ABB RobotStudio station: Lab1Station.rsstn

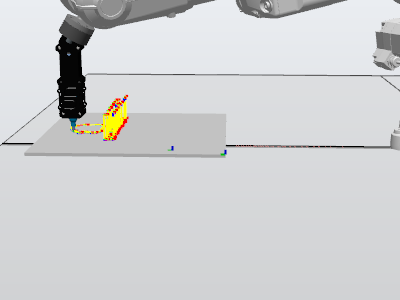
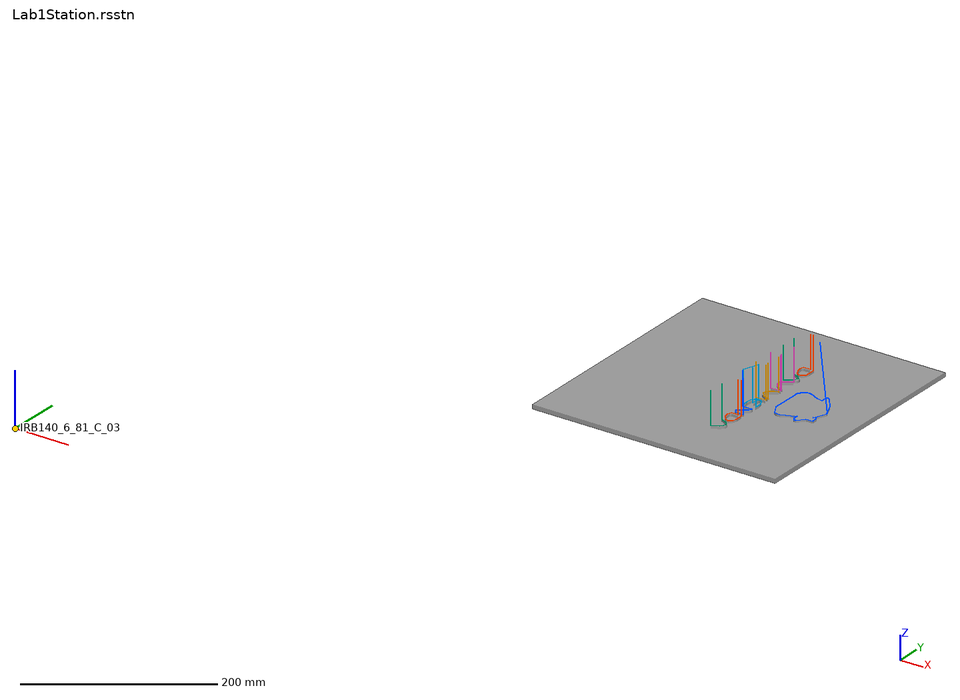
[picture v1: parts stored in the station drawn from their meshes, with robot base, taught points and paths (robot models come from the ABB library and are not in the file)]
Station Lab1Station (saved by RobotStudio 22.3.10190.2)
Controller Controller3
  mechanical unit ROB_1: IRB140_6_81_C_03, 6 joints, base frame (0, 0, 0) mm
Layout (positions relative to the parent item):
  - IRB140_6_81_C_03 [mechanism, from Robots\IRB140_6_81_C_G_03.rslib] at (0, 0, 0) mm; joint values [0.4312, 1.4172, -1.227, -0.2668, 0.9151, 0.5443] (rad or m)
  - HerrMarcador [part, from MyTools\HerrMarcadorInclinado.rslib] at (758.29, 333.88, 278.98) mm, rotated rx -180 ry 30 rz -180 deg
  - Davivienda [part] at (520, 470, 100) mm, rotated rx 0 ry 0 rz -90 deg, size 300 x 300 x 8 mm
Attachment: HerrMarcador is attached to IRB140_6_81_C_03 / Link6
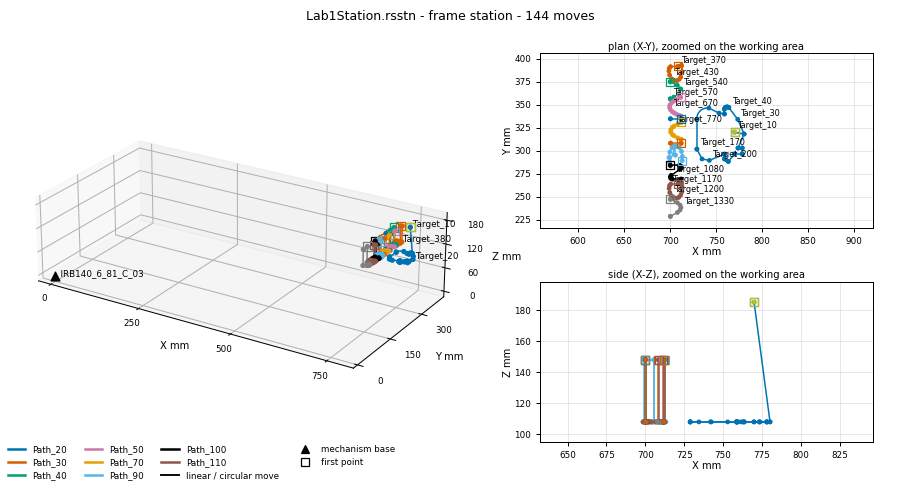
[picture p0: tool path of Lab1Station.rsstn in frame station, 144 of 146 moves have a stored position in this frame; points joined in program order, loops and branches not executed]
Targets, tools, work objects and paths stored in the station, written as RAPID:
! task T_ROB1
MODULE user
  TASK PERS tooldata Marcador_Data:=[TRUE,[[72.5,0,155.57],[0.965925826,-0.000008429,0.258819045,0.000002259]],[0.002,[19.889,-0.005,58.089],[1,0,0,0],0,0,0]];
ENDMODULE

! task T_ROB1
MODULE CalibData
  TASK PERS wobjdata Tablero:=[FALSE,TRUE,"",[[600,450,105],[0.707106781,0,0,-0.707106781]],[[-20,-80,0],[1,0,0,0]]];
ENDMODULE

! task T_ROB1
MODULE Module1
  CONST robtarget Target_10:=[[150,250,80],[0,-0.707106781,0.707106781,0],[0,-1,0,0],[9E+09,9E+09,9E+09,9E+09,9E+09,9E+09]];
  CONST robtarget Target_20:=[[152.02476718,260.252415756,3],[0,-0.707106781,0.707106781,0],[0,-1,1,0],[9E+09,9E+09,9E+09,9E+09,9E+09,9E+09]];
  CONST robtarget Target_30:=[[136.118401169,253.292570976,3],[0,-0.707106781,0.707106781,0],[0,0,0,0],[9E+09,9E+09,9E+09,9E+09,9E+09,9E+09]];
  CONST robtarget Target_40:=[[123.269606583,243.615464733,3],[0,-0.707106781,0.707106781,0],[0,-1,0,0],[9E+09,9E+09,9E+09,9E+09,9E+09,9E+09]];
  CONST robtarget Target_50:=[[123.269606583,243.615464733,3],[0,-0.707106781,0.707106781,0],[0,0,0,0],[9E+09,9E+09,9E+09,9E+09,9E+09,9E+09]];
  CONST robtarget Target_60:=[[122.281773997,241.718097026,3],[0,-0.707106781,0.707106781,0],[0,-1,0,0],[9E+09,9E+09,9E+09,9E+09,9E+09,9E+09]];
  CONST robtarget Target_70:=[[122.995762655,239.701655203,3],[0,-0.707106781,0.707106781,0],[0,0,0,0],[9E+09,9E+09,9E+09,9E+09,9E+09,9E+09]];
  CONST robtarget Target_80:=[[124.957451694,238.84866426,3],[0,-0.707106781,0.707106781,0],[0,0,0,0],[9E+09,9E+09,9E+09,9E+09,9E+09,9E+09]];
  CONST robtarget Target_90:=[[124.957451694,238.84866426,3],[0,-0.707106781,0.707106781,0],[0,0,0,0],[9E+09,9E+09,9E+09,9E+09,9E+09,9E+09]];
  CONST robtarget Target_100:=[[130.248275394,238.84866426,3],[0,-0.707106781,0.707106781,0],[0,0,0,0],[9E+09,9E+09,9E+09,9E+09,9E+09,9E+09]];
  CONST robtarget Target_110:=[[130.248275394,238.84866426,3],[0,-0.707106781,0.707106781,0],[0,0,0,0],[9E+09,9E+09,9E+09,9E+09,9E+09,9E+09]];
  CONST robtarget Target_120:=[[129.335918588,232.983108033,3],[0,-0.707106781,0.707106781,0],[0,0,0,0],[9E+09,9E+09,9E+09,9E+09,9E+09,9E+09]];
  CONST robtarget Target_130:=[[123.812362313,221.9363364,3],[0,-0.707106781,0.707106781,0],[0,0,0,0],[9E+09,9E+09,9E+09,9E+09,9E+09,9E+09]];
  CONST robtarget Target_140:=[[125.443880841,214.375036174,3],[0,-0.707106781,0.707106781,0],[0,0,0,0],[9E+09,9E+09,9E+09,9E+09,9E+09,9E+09]];
  CONST robtarget Target_150:=[[135.991781584,208.907395353,3],[0,-0.707106781,0.707106781,0],[0,0,0,0],[9E+09,9E+09,9E+09,9E+09,9E+09,9E+09]];
  CONST robtarget Target_160:=[[135.991781584,208.907395353,3],[0,-0.707106781,0.707106781,0],[0,0,0,0],[9E+09,9E+09,9E+09,9E+09,9E+09,9E+09]];
  CONST robtarget Target_170:=[[168.476558528,208.907395353,3],[0,-0.707106781,0.707106781,0],[0,0,0,0],[9E+09,9E+09,9E+09,9E+09,9E+09,9E+09]];
  CONST robtarget Target_180:=[[168.476558528,208.907395353,3],[0,-0.707106781,0.707106781,0],[0,0,0,0],[9E+09,9E+09,9E+09,9E+09,9E+09,9E+09]];
  CONST robtarget Target_190:=[[179.114572542,214.493962129,3],[0,-0.707106781,0.707106781,0],[0,0,0,0],[9E+09,9E+09,9E+09,9E+09,9E+09,9E+09]];
  CONST robtarget Target_200:=[[180.686258584,222.455286023,3],[0,-0.707106781,0.707106781,0],[0,0,0,0],[9E+09,9E+09,9E+09,9E+09,9E+09,9E+09]];
  CONST robtarget Target_210:=[[173.93550103,238.84866426,3],[0,-0.707106781,0.707106781,0],[0,0,0,0],[9E+09,9E+09,9E+09,9E+09,9E+09,9E+09]];
  CONST robtarget Target_220:=[[173.93550103,238.84866426,3],[0,-0.707106781,0.707106781,0],[0,0,0,0],[9E+09,9E+09,9E+09,9E+09,9E+09,9E+09]];
  CONST robtarget Target_230:=[[179.092082666,238.84866426,3],[0,-0.707106781,0.707106781,0],[0,0,0,0],[9E+09,9E+09,9E+09,9E+09,9E+09,9E+09]];
  CONST robtarget Target_240:=[[179.092082666,238.84866426,3],[0,-0.707106781,0.707106781,0],[0,0,0,0],[9E+09,9E+09,9E+09,9E+09,9E+09,9E+09]];
  CONST robtarget Target_250:=[[181.598076735,240.213820445,3],[0,-0.707106781,0.707106781,0],[0,0,0,0],[9E+09,9E+09,9E+09,9E+09,9E+09,9E+09]];
  CONST robtarget Target_260:=[[181.810114173,243.059641558,3],[0,-0.707106781,0.707106781,0],[0,0,0,0],[9E+09,9E+09,9E+09,9E+09,9E+09,9E+09]];
  CONST robtarget Target_270:=[[181.810114173,243.059641558,3],[0,-0.707106781,0.707106781,0],[0,0,0,0],[9E+09,9E+09,9E+09,9E+09,9E+09,9E+09]];
  CONST robtarget Target_280:=[[173.790831816,249.924383369,3],[0,-0.707106781,0.707106781,0],[0,0,0,0],[9E+09,9E+09,9E+09,9E+09,9E+09,9E+09]];
  CONST robtarget Target_290:=[[173.790831816,249.924383369,3],[0,-0.707106781,0.707106781,0],[0,0,0,0],[9E+09,9E+09,9E+09,9E+09,9E+09,9E+09]];
  CONST robtarget Target_300:=[[173.790831816,258.182639544,3],[0,-0.707106781,0.707106781,0],[0,0,0,0],[9E+09,9E+09,9E+09,9E+09,9E+09,9E+09]];
  CONST robtarget Target_310:=[[173.790831816,258.182639544,3],[0,-0.707106781,0.707106781,0],[0,0,0,0],[9E+09,9E+09,9E+09,9E+09,9E+09,9E+09]];
  CONST robtarget Target_320:=[[167.241395906,258.182639544,3],[0,-0.707106781,0.707106781,0],[0,0,0,0],[9E+09,9E+09,9E+09,9E+09,9E+09,9E+09]];
  CONST robtarget Target_330:=[[167.241395906,258.182639544,3],[0,-0.707106781,0.707106781,0],[0,0,0,0],[9E+09,9E+09,9E+09,9E+09,9E+09,9E+09]];
  CONST robtarget Target_340:=[[167.241395906,253.645994177,3],[0,-0.707106781,0.707106781,0],[0,0,0,0],[9E+09,9E+09,9E+09,9E+09,9E+09,9E+09]];
  CONST robtarget Target_350:=[[167.241395906,253.645994177,3],[0,-0.707106781,0.707106781,0],[0,0,0,0],[9E+09,9E+09,9E+09,9E+09,9E+09,9E+09]];
  CONST robtarget Target_360:=[[152.02476718,260.252415756,3],[0,-0.707106781,0.707106781,0],[0,0,0,0],[9E+09,9E+09,9E+09,9E+09,9E+09,9E+09]];
  CONST robtarget Target_370:=[[78.556394934,188.285452755,43],[0,-0.707106781,0.707106781,0],[0,0,0,0],[9E+09,9E+09,9E+09,9E+09,9E+09,9E+09]];
  CONST robtarget Target_380:=[[78.556394934,188.285452755,3],[0,-0.707106781,0.707106781,0],[0,0,0,0],[9E+09,9E+09,9E+09,9E+09,9E+09,9E+09]];
  CONST robtarget Target_390:=[[78.777217091,180.337746759,3],[0,-0.707106781,0.707106781,0],[0,0,0,0],[9E+09,9E+09,9E+09,9E+09,9E+09,9E+09]];
  CONST robtarget Target_400:=[[80.371798013,178.989551395,3],[0,-0.707106781,0.707106781,0],[0,0,0,0],[9E+09,9E+09,9E+09,9E+09,9E+09,9E+09]];
  CONST robtarget Target_410:=[[83.506257563,178.489977672,3],[0,-0.707106781,0.707106781,0],[0,0,0,0],[9E+09,9E+09,9E+09,9E+09,9E+09,9E+09]];
  CONST robtarget Target_420:=[[87.997557508,179.252868031,3],[0,-0.707106781,0.707106781,0],[0,0,0,0],[9E+09,9E+09,9E+09,9E+09,9E+09,9E+09]];
  CONST robtarget Target_430:=[[92.028971208,181.53752069,3],[0,-0.707106781,0.707106781,0],[0,0,0,0],[9E+09,9E+09,9E+09,9E+09,9E+09,9E+09]];
  CONST robtarget Target_440:=[[93.868246154,184.336737299,3],[0,-0.707106781,0.707106781,0],[0,0,0,0],[9E+09,9E+09,9E+09,9E+09,9E+09,9E+09]];
  CONST robtarget Target_450:=[[94.007732668,187.144143926,3],[0,-0.707106781,0.707106781,0],[0,0,0,0],[9E+09,9E+09,9E+09,9E+09,9E+09,9E+09]];
  CONST robtarget Target_460:=[[92.604060403,189.719708823,3],[0,-0.707106781,0.707106781,0],[0,0,0,0],[9E+09,9E+09,9E+09,9E+09,9E+09,9E+09]];
  CONST robtarget Target_470:=[[90.06132568,191.417144488,3],[0,-0.707106781,0.707106781,0],[0,0,0,0],[9E+09,9E+09,9E+09,9E+09,9E+09,9E+09]];
  CONST robtarget Target_480:=[[85.079316563,192.471582305,3],[0,-0.707106781,0.707106781,0],[0,0,0,0],[9E+09,9E+09,9E+09,9E+09,9E+09,9E+09]];
  CONST robtarget Target_490:=[[77.598246493,192.118931644,3],[0,-0.707106781,0.707106781,0],[0,0,0,0],[9E+09,9E+09,9E+09,9E+09,9E+09,9E+09]];
  CONST robtarget Target_500:=[[77.598246493,192.118931644,43],[0,-0.707106781,0.707106781,0],[0,0,0,0],[9E+09,9E+09,9E+09,9E+09,9E+09,9E+09]];
  CONST robtarget Target_510:=[[95.28667285,179.972658622,43],[0,-0.707106781,0.707106781,0],[0,0,0,0],[9E+09,9E+09,9E+09,9E+09,9E+09,9E+09]];
  CONST robtarget Target_520:=[[95.28667285,179.972658622,3],[0,-0.707106781,0.707106781,0],[0,0,0,0],[9E+09,9E+09,9E+09,9E+09,9E+09,9E+09]];
  CONST robtarget Target_530:=[[99.054803913,187.648232468,3],[0,-0.707106781,0.707106781,0],[0,0,0,0],[9E+09,9E+09,9E+09,9E+09,9E+09,9E+09]];
  CONST robtarget Target_540:=[[102.919910411,191.254451105,3],[0,-0.707106781,0.707106781,0],[0,0,0,0],[9E+09,9E+09,9E+09,9E+09,9E+09,9E+09]];
  CONST robtarget Target_550:=[[108.350570105,189.25957291,3],[0,-0.707106781,0.707106781,0],[0,0,0,0],[9E+09,9E+09,9E+09,9E+09,9E+09,9E+09]];
  CONST robtarget Target_560:=[[111.949527633,183.734460812,3],[0,-0.707106781,0.707106781,0],[0,0,0,0],[9E+09,9E+09,9E+09,9E+09,9E+09,9E+09]];
  CONST robtarget Target_570:=[[113.857897554,179.972658622,3],[0,-0.707106781,0.707106781,0],[0,0,0,0],[9E+09,9E+09,9E+09,9E+09,9E+09,9E+09]];
  CONST robtarget Target_580:=[[113.857897554,179.972658622,43],[0,-0.707106781,0.707106781,0],[0,0,0,0],[9E+09,9E+09,9E+09,9E+09,9E+09,9E+09]];
  CONST robtarget Target_590:=[[112.126063194,191.2423046,43],[0,-0.707106781,0.707106781,0],[0,0,0,0],[9E+09,9E+09,9E+09,9E+09,9E+09,9E+09]];
  CONST robtarget Target_600:=[[112.126063194,191.2423046,3],[0,-0.707106781,0.707106781,0],[0,0,0,0],[9E+09,9E+09,9E+09,9E+09,9E+09,9E+09]];
  CONST robtarget Target_610:=[[114.401889485,186.789312293,3],[0,-0.707106781,0.707106781,0],[0,0,0,0],[9E+09,9E+09,9E+09,9E+09,9E+09,9E+09]];
  CONST robtarget Target_620:=[[115.58057196,184.74123642,3],[0,-0.707106781,0.707106781,0],[0,0,0,0],[9E+09,9E+09,9E+09,9E+09,9E+09,9E+09]];
  CONST robtarget Target_630:=[[116.864504777,182.854229079,3],[0,-0.707106781,0.707106781,0],[0,0,0,0],[9E+09,9E+09,9E+09,9E+09,9E+09,9E+09]];
  CONST robtarget Target_640:=[[118.25426578,181.252000645,3],[0,-0.707106781,0.707106781,0],[0,0,0,0],[9E+09,9E+09,9E+09,9E+09,9E+09,9E+09]];
  CONST robtarget Target_650:=[[120.57420176,179.604352291,3],[0,-0.707106781,0.707106781,0],[0,0,0,0],[9E+09,9E+09,9E+09,9E+09,9E+09,9E+09]];
  CONST robtarget Target_660:=[[123.164632355,179.201937245,3],[0,-0.707106781,0.707106781,0],[0,0,0,0],[9E+09,9E+09,9E+09,9E+09,9E+09,9E+09]];
  CONST robtarget Target_670:=[[125.643689482,180.211828512,3],[0,-0.707106781,0.707106781,0],[0,0,0,0],[9E+09,9E+09,9E+09,9E+09,9E+09,9E+09]];
  CONST robtarget Target_680:=[[127.787428256,182.296804988,3],[0,-0.707106781,0.707106781,0],[0,0,0,0],[9E+09,9E+09,9E+09,9E+09,9E+09,9E+09]];
  CONST robtarget Target_690:=[[129.053529141,184.108665847,3],[0,-0.707106781,0.707106781,0],[0,0,0,0],[9E+09,9E+09,9E+09,9E+09,9E+09,9E+09]];
  CONST robtarget Target_700:=[[130.193418821,186.12829205,3],[0,-0.707106781,0.707106781,0],[0,0,0,0],[9E+09,9E+09,9E+09,9E+09,9E+09,9E+09]];
  CONST robtarget Target_710:=[[131.496798753,188.892443357,3],[0,-0.707106781,0.707106781,0],[0,0,0,0],[9E+09,9E+09,9E+09,9E+09,9E+09,9E+09]];
  CONST robtarget Target_720:=[[132.509994829,191.333655407,3],[0,-0.707106781,0.707106781,0],[0,0,0,0],[9E+09,9E+09,9E+09,9E+09,9E+09,9E+09]];
  CONST robtarget Target_730:=[[132.509994829,191.333655407,43],[0,-0.707106781,0.707106781,0],[0,0,0,0],[9E+09,9E+09,9E+09,9E+09,9E+09,9E+09]];
  CONST robtarget Target_850:=[[157.76203271,191.808660142,43],[0,-0.707106781,0.707106781,0],[0,0,0,0],[9E+09,9E+09,9E+09,9E+09,9E+09,9E+09]];
  CONST robtarget Target_840:=[[157.76203271,191.808660142,3],[0,-0.707106781,0.707106781,0],[0,0,0,0],[9E+09,9E+09,9E+09,9E+09,9E+09,9E+09]];
  CONST robtarget Target_830:=[[156.15234039,188.046857953,3],[0,-0.707106781,0.707106781,0],[0,0,0,0],[9E+09,9E+09,9E+09,9E+09,9E+09,9E+09]];
  CONST robtarget Target_820:=[[153.993901647,184.133086296,3],[0,-0.707106781,0.707106781,0],[0,0,0,0],[9E+09,9E+09,9E+09,9E+09,9E+09,9E+09]];
  CONST robtarget Target_810:=[[152.767003941,182.521745854,3],[0,-0.707106781,0.707106781,0],[0,0,0,0],[9E+09,9E+09,9E+09,9E+09,9E+09,9E+09]];
  CONST robtarget Target_800:=[[150.12879515,180.526867659,3],[0,-0.707106781,0.707106781,0],[0,0,0,0],[9E+09,9E+09,9E+09,9E+09,9E+09,9E+09]];
  CONST robtarget Target_790:=[[147.385613086,180.526867659,3],[0,-0.707106781,0.707106781,0],[0,0,0,0],[9E+09,9E+09,9E+09,9E+09,9E+09,9E+09]];
  CONST robtarget Target_780:=[[144.698135455,182.521745854,3],[0,-0.707106781,0.707106781,0],[0,0,0,0],[9E+09,9E+09,9E+09,9E+09,9E+09,9E+09]];
  CONST robtarget Target_770:=[[143.422867655,184.133086296,3],[0,-0.707106781,0.707106781,0],[0,0,0,0],[9E+09,9E+09,9E+09,9E+09,9E+09,9E+09]];
  CONST robtarget Target_760:=[[141.099177927,188.046857953,3],[0,-0.707106781,0.707106781,0],[0,0,0,0],[9E+09,9E+09,9E+09,9E+09,9E+09,9E+09]];
  CONST robtarget Target_750:=[[139.190808007,191.808660142,3],[0,-0.707106781,0.707106781,0],[0,0,0,0],[9E+09,9E+09,9E+09,9E+09,9E+09,9E+09]];
  CONST robtarget Target_740:=[[139.190808007,191.808660142,43],[0,-0.707106781,0.707106781,0],[0,0,0,0],[9E+09,9E+09,9E+09,9E+09,9E+09,9E+09]];
  CONST robtarget Target_860:=[[180.900017621,192.772598931,43],[0,-0.707106781,0.707106781,0],[0,0,0,0],[9E+09,9E+09,9E+09,9E+09,9E+09,9E+09]];
  CONST robtarget Target_870:=[[180.900017621,192.772598931,3],[0,-0.707106781,0.707106781,0],[0,0,0,0],[9E+09,9E+09,9E+09,9E+09,9E+09,9E+09]];
  CONST robtarget Target_880:=[[176.382939367,193.212871714,3],[0,-0.707106781,0.707106781,0],[0,0,0,0],[9E+09,9E+09,9E+09,9E+09,9E+09,9E+09]];
  CONST robtarget Target_890:=[[170.970258042,192.198847376,3],[0,-0.707106781,0.707106781,0],[0,0,0,0],[9E+09,9E+09,9E+09,9E+09,9E+09,9E+09]];
  CONST robtarget Target_900:=[[166.785952121,189.888900617,3],[0,-0.707106781,0.707106781,0],[0,0,0,0],[9E+09,9E+09,9E+09,9E+09,9E+09,9E+09]];
  CONST robtarget Target_910:=[[164.952754986,187.114242389,3],[0,-0.707106781,0.707106781,0],[0,0,0,0],[9E+09,9E+09,9E+09,9E+09,9E+09,9E+09]];
  CONST robtarget Target_920:=[[165.164721282,184.270843116,3],[0,-0.707106781,0.707106781,0],[0,0,0,0],[9E+09,9E+09,9E+09,9E+09,9E+09,9E+09]];
  CONST robtarget Target_930:=[[167.093724566,181.809257284,3],[0,-0.707106781,0.707106781,0],[0,0,0,0],[9E+09,9E+09,9E+09,9E+09,9E+09,9E+09]];
  CONST robtarget Target_940:=[[171.616042828,179.471063414,3],[0,-0.707106781,0.707106781,0],[0,0,0,0],[9E+09,9E+09,9E+09,9E+09,9E+09,9E+09]];
  CONST robtarget Target_950:=[[177.570763361,178.558209179,3],[0,-0.707106781,0.707106781,0],[0,0,0,0],[9E+09,9E+09,9E+09,9E+09,9E+09,9E+09]];
  CONST robtarget Target_960:=[[182.739143883,179.363545337,3],[0,-0.707106781,0.707106781,0],[0,0,0,0],[9E+09,9E+09,9E+09,9E+09,9E+09,9E+09]];
  CONST robtarget Target_970:=[[182.739143883,179.363545337,43],[0,-0.707106781,0.707106781,0],[0,0,0,0],[9E+09,9E+09,9E+09,9E+09,9E+09,9E+09]];
  CONST robtarget Target_980:=[[165.856491279,185.425872658,43],[0,-0.707106781,0.707106781,0],[0,0,0,0],[9E+09,9E+09,9E+09,9E+09,9E+09,9E+09]];
  CONST robtarget Target_990:=[[165.856491279,185.425872658,3],[0,-0.707106781,0.707106781,0],[0,0,0,0],[9E+09,9E+09,9E+09,9E+09,9E+09,9E+09]];
  CONST robtarget Target_1000:=[[174.881326239,185.425872658,3],[0,-0.707106781,0.707106781,0],[0,0,0,0],[9E+09,9E+09,9E+09,9E+09,9E+09,9E+09]];
  CONST robtarget Target_1010:=[[174.881326239,185.425872658,43],[0,-0.707106781,0.707106781,0],[0,0,0,0],[9E+09,9E+09,9E+09,9E+09,9E+09,9E+09]];
  CONST robtarget Target_1020:=[[186.056975108,180.0240886,43],[0,-0.707106781,0.707106781,0],[0,0,0,0],[9E+09,9E+09,9E+09,9E+09,9E+09,9E+09]];
  CONST robtarget Target_1030:=[[186.056975108,180.0240886,3],[0,-0.707106781,0.707106781,0],[0,0,0,0],[9E+09,9E+09,9E+09,9E+09,9E+09,9E+09]];
  CONST robtarget Target_1040:=[[186.056975108,189.935023093,3],[0,-0.707106781,0.707106781,0],[0,0,0,0],[9E+09,9E+09,9E+09,9E+09,9E+09,9E+09]];
  CONST robtarget Target_1050:=[[186.763325262,191.505223547,3],[0,-0.707106781,0.707106781,0],[0,0,0,0],[9E+09,9E+09,9E+09,9E+09,9E+09,9E+09]];
  CONST robtarget Target_1060:=[[188.406849438,192.018339801,3],[0,-0.707106781,0.707106781,0],[0,0,0,0],[9E+09,9E+09,9E+09,9E+09,9E+09,9E+09]];
  CONST robtarget Target_1070:=[[189.881100727,191.128933739,3],[0,-0.707106781,0.707106781,0],[0,0,0,0],[9E+09,9E+09,9E+09,9E+09,9E+09,9E+09]];
  CONST robtarget Target_1080:=[[197.020438855,180.996681372,3],[0,-0.707106781,0.707106781,0],[0,0,0,0],[9E+09,9E+09,9E+09,9E+09,9E+09,9E+09]];
  CONST robtarget Target_1090:=[[198.546692612,180.070671426,3],[0,-0.707106781,0.707106781,0],[0,0,0,0],[9E+09,9E+09,9E+09,9E+09,9E+09,9E+09]];
  CONST robtarget Target_1100:=[[200.263393096,180.560451375,3],[0,-0.707106781,0.707106781,0],[0,0,0,0],[9E+09,9E+09,9E+09,9E+09,9E+09,9E+09]];
  CONST robtarget Target_1110:=[[201.071266889,182.15239512,3],[0,-0.707106781,0.707106781,0],[0,0,0,0],[9E+09,9E+09,9E+09,9E+09,9E+09,9E+09]];
  CONST robtarget Target_1120:=[[201.071266889,191.808458708,3],[0,-0.707106781,0.707106781,0],[0,0,0,0],[9E+09,9E+09,9E+09,9E+09,9E+09,9E+09]];
  CONST robtarget Target_1130:=[[201.071266889,191.808458708,43],[0,-0.707106781,0.707106781,0],[0,0,0,0],[9E+09,9E+09,9E+09,9E+09,9E+09,9E+09]];
  CONST robtarget Target_1140:=[[206.229553228,188.507024825,43],[0,-0.707106781,0.707106781,0],[0,0,0,0],[9E+09,9E+09,9E+09,9E+09,9E+09,9E+09]];
  CONST robtarget Target_1150:=[[206.229553228,188.507024825,3],[0,-0.707106781,0.707106781,0],[0,0,0,0],[9E+09,9E+09,9E+09,9E+09,9E+09,9E+09]];
  CONST robtarget Target_1160:=[[206.450375385,180.559318829,3],[0,-0.707106781,0.707106781,0],[0,0,0,0],[9E+09,9E+09,9E+09,9E+09,9E+09,9E+09]];
  CONST robtarget Target_1170:=[[208.044956306,179.211123465,3],[0,-0.707106781,0.707106781,0],[0,0,0,0],[9E+09,9E+09,9E+09,9E+09,9E+09,9E+09]];
  CONST robtarget Target_1180:=[[211.179415856,178.711549742,3],[0,-0.707106781,0.707106781,0],[0,0,0,0],[9E+09,9E+09,9E+09,9E+09,9E+09,9E+09]];
  CONST robtarget Target_1190:=[[215.670715802,179.474440101,3],[0,-0.707106781,0.707106781,0],[0,0,0,0],[9E+09,9E+09,9E+09,9E+09,9E+09,9E+09]];
  CONST robtarget Target_1200:=[[219.146674086,181.285925923,3],[0,-0.707106781,0.707106781,0],[0,0,0,0],[9E+09,9E+09,9E+09,9E+09,9E+09,9E+09]];
  CONST robtarget Target_1210:=[[221.167303294,183.657599156,3],[0,-0.707106781,0.707106781,0],[0,0,0,0],[9E+09,9E+09,9E+09,9E+09,9E+09,9E+09]];
  CONST robtarget Target_1220:=[[221.802063231,186.429372352,3],[0,-0.707106781,0.707106781,0],[0,0,0,0],[9E+09,9E+09,9E+09,9E+09,9E+09,9E+09]];
  CONST robtarget Target_1230:=[[220.918759188,189.142114999,3],[0,-0.707106781,0.707106781,0],[0,0,0,0],[9E+09,9E+09,9E+09,9E+09,9E+09,9E+09]];
  CONST robtarget Target_1240:=[[218.483605633,191.280183866,3],[0,-0.707106781,0.707106781,0],[0,0,0,0],[9E+09,9E+09,9E+09,9E+09,9E+09,9E+09]];
  CONST robtarget Target_1250:=[[215.007692517,192.425603275,3],[0,-0.707106781,0.707106781,0],[0,0,0,0],[9E+09,9E+09,9E+09,9E+09,9E+09,9E+09]];
  CONST robtarget Target_1260:=[[208.610688293,192.668819455,3],[0,-0.707106781,0.707106781,0],[0,0,0,0],[9E+09,9E+09,9E+09,9E+09,9E+09,9E+09]];
  CONST robtarget Target_1270:=[[205.271404786,192.340503714,3],[0,-0.707106781,0.707106781,0],[0,0,0,0],[9E+09,9E+09,9E+09,9E+09,9E+09,9E+09]];
  CONST robtarget Target_1280:=[[205.271404786,192.340503714,43],[0,-0.707106781,0.707106781,0],[0,0,0,0],[9E+09,9E+09,9E+09,9E+09,9E+09,9E+09]];
  CONST robtarget Target_1290:=[[222.942235464,180.076706447,43],[0,-0.707106781,0.707106781,0],[0,0,0,0],[9E+09,9E+09,9E+09,9E+09,9E+09,9E+09]];
  CONST robtarget Target_1300:=[[222.942235464,180.076706447,3],[0,-0.707106781,0.707106781,0],[0,0,0,0],[9E+09,9E+09,9E+09,9E+09,9E+09,9E+09]];
  CONST robtarget Target_1310:=[[226.710366527,187.752280293,3],[0,-0.707106781,0.707106781,0],[0,0,0,0],[9E+09,9E+09,9E+09,9E+09,9E+09,9E+09]];
  CONST robtarget Target_1320:=[[229.232828908,190.591251324,3],[0,-0.707106781,0.707106781,0],[0,0,0,0],[9E+09,9E+09,9E+09,9E+09,9E+09,9E+09]];
  CONST robtarget Target_1330:=[[231.944210176,191.619359674,3],[0,-0.707106781,0.707106781,0],[0,0,0,0],[9E+09,9E+09,9E+09,9E+09,9E+09,9E+09]];
  CONST robtarget Target_1340:=[[234.679023609,190.591251324,3],[0,-0.707106781,0.707106781,0],[0,0,0,0],[9E+09,9E+09,9E+09,9E+09,9E+09,9E+09]];
  CONST robtarget Target_1350:=[[237.281400519,187.752280293,3],[0,-0.707106781,0.707106781,0],[0,0,0,0],[9E+09,9E+09,9E+09,9E+09,9E+09,9E+09]];
  CONST robtarget Target_1360:=[[241.513460167,180.076706447,3],[0,-0.707106781,0.707106781,0],[0,0,0,0],[9E+09,9E+09,9E+09,9E+09,9E+09,9E+09]];
  CONST robtarget Target_1370:=[[241.513460167,180.076706447,43],[0,-0.707106781,0.707106781,0],[0,0,0,0],[9E+09,9E+09,9E+09,9E+09,9E+09,9E+09]];
  CONST jointtarget JointTarget_1:=[[0,0,0,0,30,0],[9E+09,9E+09,9E+09,9E+09,9E+09,9E+09]];
  CONST jointtarget JointTarget_2:=[[90,0,0,0,-60,0],[9E+09,9E+09,9E+09,9E+09,9E+09,9E+09]];
  CONST robtarget Target_1380:=[[135.514873091,191.707491867,43],[0,-0.707106781,0.707106781,0],[0,0,0,0],[9E+09,9E+09,9E+09,9E+09,9E+09,9E+09]];
  CONST robtarget Target_1390:=[[135.514873091,191.707491867,3],[0,-0.707106781,0.707106781,0],[0,0,0,0],[9E+09,9E+09,9E+09,9E+09,9E+09,9E+09]];
  CONST robtarget Target_1400:=[[135.514873091,180.207491867,3],[0,-0.707106781,0.707106781,0],[0,0,0,0],[9E+09,9E+09,9E+09,9E+09,9E+09,9E+09]];
  CONST robtarget Target_1410:=[[135.514873091,180.207491867,43],[0,-0.707106781,0.707106781,0],[0,0,0,0],[9E+09,9E+09,9E+09,9E+09,9E+09,9E+09]];
  CONST robtarget Target_1420:=[[162.001803873,191.808458708,43],[0,-0.707106781,0.707106781,0],[0,0,0,0],[9E+09,9E+09,9E+09,9E+09,9E+09,9E+09]];
  CONST robtarget Target_1430:=[[162.001803873,191.808458708,3],[0,-0.707106781,0.707106781,0],[0,0,0,0],[9E+09,9E+09,9E+09,9E+09,9E+09,9E+09]];
  CONST robtarget Target_1440:=[[162.001803873,180.308458708,3],[0,-0.707106781,0.707106781,0],[0,0,0,0],[9E+09,9E+09,9E+09,9E+09,9E+09,9E+09]];
  CONST robtarget Target_1450:=[[162.001803873,180.308458708,43],[0,-0.707106781,0.707106781,0],[0,0,0,0],[9E+09,9E+09,9E+09,9E+09,9E+09,9E+09]];
  PROC Path_20()
    MoveL Target_10,v100,z5,Marcador_Data\WObj:=Tablero;
    MoveL Target_20,v100,z5,Marcador_Data\WObj:=Tablero;
    MoveL Target_30,v100,z5,Marcador_Data\WObj:=Tablero;
    MoveL Target_40,v100,z5,Marcador_Data\WObj:=Tablero;
    MoveL Target_50,v100,z5,Marcador_Data\WObj:=Tablero;
    MoveL Target_60,v100,z5,Marcador_Data\WObj:=Tablero;
    MoveL Target_70,v100,z5,Marcador_Data\WObj:=Tablero;
    MoveL Target_80,v100,z5,Marcador_Data\WObj:=Tablero;
    MoveL Target_90,v100,z5,Marcador_Data\WObj:=Tablero;
    MoveL Target_100,v100,z5,Marcador_Data\WObj:=Tablero;
    MoveL Target_110,v100,z5,Marcador_Data\WObj:=Tablero;
    MoveL Target_120,v100,z5,Marcador_Data\WObj:=Tablero;
    MoveL Target_130,v100,z5,Marcador_Data\WObj:=Tablero;
    MoveC Target_140,Target_150,v100,z5,Marcador_Data\WObj:=Tablero;
    MoveL Target_160,v100,z5,Marcador_Data\WObj:=Tablero;
    MoveL Target_170,v100,z5,Marcador_Data\WObj:=Tablero;
    MoveL Target_180,v100,z5,Marcador_Data\WObj:=Tablero;
    MoveL Target_190,v100,z5,Marcador_Data\WObj:=Tablero;
    MoveL Target_200,v100,z5,Marcador_Data\WObj:=Tablero;
    MoveL Target_210,v100,z5,Marcador_Data\WObj:=Tablero;
    MoveL Target_220,v100,z5,Marcador_Data\WObj:=Tablero;
    MoveL Target_230,v100,z5,Marcador_Data\WObj:=Tablero;
    MoveL Target_240,v100,z5,Marcador_Data\WObj:=Tablero;
    MoveC Target_250,Target_260,v100,z5,Marcador_Data\WObj:=Tablero;
    MoveL Target_270,v100,z5,Marcador_Data\WObj:=Tablero;
    MoveL Target_280,v100,z5,Marcador_Data\WObj:=Tablero;
    MoveL Target_290,v100,z5,Marcador_Data\WObj:=Tablero;
    MoveL Target_300,v100,z5,Marcador_Data\WObj:=Tablero;
    MoveL Target_310,v100,z5,Marcador_Data\WObj:=Tablero;
    MoveL Target_320,v100,z5,Marcador_Data\WObj:=Tablero;
    MoveL Target_330,v100,z5,Marcador_Data\WObj:=Tablero;
    MoveL Target_340,v100,z5,Marcador_Data\WObj:=Tablero;
    MoveL Target_350,v100,z5,Marcador_Data\WObj:=Tablero;
    MoveL Target_360,v100,z5,Marcador_Data\WObj:=Tablero;
  ENDPROC
  PROC main()
    SetDO DO_02,0;
    Path_10;
    SetDO DO_01,1;
    Path_20;
    Path_30;
    Path_40;
    Path_50;
    Path_60;
    Path_70;
    Path_80;
    Path_90;
    Path_100;
    Path_110;
    Path_120;
    Path_130;
    SetDO DO_01,0;
    Path_10;
    SetDO DO_02,1;
    Path_140;
  ENDPROC
  PROC Path_30()
    MoveL Target_370,v100,z5,Marcador_Data\WObj:=Tablero;
    MoveL Target_380,v100,z5,Marcador_Data\WObj:=Tablero;
    MoveL Target_390,v100,z5,Marcador_Data\WObj:=Tablero;
    MoveL Target_400,v100,z5,Marcador_Data\WObj:=Tablero;
    MoveL Target_410,v100,z5,Marcador_Data\WObj:=Tablero;
    MoveL Target_420,v100,z5,Marcador_Data\WObj:=Tablero;
    MoveL Target_430,v100,z5,Marcador_Data\WObj:=Tablero;
    MoveL Target_440,v100,z5,Marcador_Data\WObj:=Tablero;
    MoveL Target_450,v100,z5,Marcador_Data\WObj:=Tablero;
    MoveL Target_460,v100,z5,Marcador_Data\WObj:=Tablero;
    MoveL Target_470,v100,z5,Marcador_Data\WObj:=Tablero;
    MoveL Target_480,v100,z5,Marcador_Data\WObj:=Tablero;
    MoveL Target_490,v100,z5,Marcador_Data\WObj:=Tablero;
    MoveL Target_500,v100,z5,Marcador_Data\WObj:=Tablero;
  ENDPROC
  PROC Path_40()
    MoveL Target_510,v100,z5,Marcador_Data\WObj:=Tablero;
    MoveL Target_520,v100,z5,Marcador_Data\WObj:=Tablero;
    MoveL Target_530,v100,z5,Marcador_Data\WObj:=Tablero;
    MoveL Target_540,v100,z5,Marcador_Data\WObj:=Tablero;
    MoveL Target_550,v100,z5,Marcador_Data\WObj:=Tablero;
    MoveL Target_560,v100,z5,Marcador_Data\WObj:=Tablero;
    MoveL Target_570,v100,z5,Marcador_Data\WObj:=Tablero;
    MoveL Target_580,v100,z5,Marcador_Data\WObj:=Tablero;
  ENDPROC
  PROC Path_50()
    MoveL Target_590,v100,z5,Marcador_Data\WObj:=Tablero;
    MoveL Target_600,v100,z5,Marcador_Data\WObj:=Tablero;
    MoveL Target_610,v100,z5,Marcador_Data\WObj:=Tablero;
    MoveL Target_620,v100,z5,Marcador_Data\WObj:=Tablero;
    MoveL Target_630,v100,z5,Marcador_Data\WObj:=Tablero;
    MoveL Target_640,v100,z5,Marcador_Data\WObj:=Tablero;
    MoveL Target_650,v100,z5,Marcador_Data\WObj:=Tablero;
    MoveL Target_660,v100,z5,Marcador_Data\WObj:=Tablero;
    MoveL Target_670,v100,z5,Marcador_Data\WObj:=Tablero;
    MoveL Target_680,v100,z5,Marcador_Data\WObj:=Tablero;
    MoveL Target_690,v100,z5,Marcador_Data\WObj:=Tablero;
    MoveL Target_700,v100,z5,Marcador_Data\WObj:=Tablero;
    MoveL Target_710,v100,z5,Marcador_Data\WObj:=Tablero;
    MoveL Target_720,v100,z5,Marcador_Data\WObj:=Tablero;
    MoveL Target_730,v100,z5,Marcador_Data\WObj:=Tablero;
  ENDPROC
  PROC Path_70()
    MoveL Target_740,v100,z5,Marcador_Data\WObj:=Tablero;
    MoveL Target_750,v100,z5,Marcador_Data\WObj:=Tablero;
    MoveL Target_760,v100,z5,Marcador_Data\WObj:=Tablero;
    MoveL Target_770,v100,z5,Marcador_Data\WObj:=Tablero;
    MoveL Target_780,v100,z5,Marcador_Data\WObj:=Tablero;
    MoveL Target_790,v100,z5,Marcador_Data\WObj:=Tablero;
    MoveL Target_800,v100,z5,Marcador_Data\WObj:=Tablero;
    MoveL Target_810,v100,z5,Marcador_Data\WObj:=Tablero;
    MoveL Target_820,v100,z5,Marcador_Data\WObj:=Tablero;
    MoveL Target_830,v100,z5,Marcador_Data\WObj:=Tablero;
    MoveL Target_840,v100,z5,Marcador_Data\WObj:=Tablero;
    MoveL Target_850,v100,z5,Marcador_Data\WObj:=Tablero;
  ENDPROC
  PROC Path_90()
    MoveL Target_860,v100,z5,Marcador_Data\WObj:=Tablero;
    MoveL Target_870,v100,z5,Marcador_Data\WObj:=Tablero;
    MoveL Target_880,v100,z5,Marcador_Data\WObj:=Tablero;
    MoveL Target_890,v100,z5,Marcador_Data\WObj:=Tablero;
    MoveL Target_900,v100,z5,Marcador_Data\WObj:=Tablero;
    MoveL Target_910,v100,z5,Marcador_Data\WObj:=Tablero;
    MoveL Target_920,v100,z5,Marcador_Data\WObj:=Tablero;
    MoveL Target_930,v100,z5,Marcador_Data\WObj:=Tablero;
    MoveL Target_940,v100,z5,Marcador_Data\WObj:=Tablero;
    MoveL Target_950,v100,z5,Marcador_Data\WObj:=Tablero;
    MoveL Target_960,v100,z5,Marcador_Data\WObj:=Tablero;
    MoveL Target_970,v100,z5,Marcador_Data\WObj:=Tablero;
    MoveL Target_980,v100,z5,Marcador_Data\WObj:=Tablero;
    MoveL Target_990,v100,z5,Marcador_Data\WObj:=Tablero;
    MoveL Target_1000,v100,z5,Marcador_Data\WObj:=Tablero;
    MoveL Target_1010,v100,z5,Marcador_Data\WObj:=Tablero;
  ENDPROC
  PROC Path_100()
    MoveL Target_1020,v100,z5,Marcador_Data\WObj:=Tablero;
    MoveL Target_1030,v100,z5,Marcador_Data\WObj:=Tablero;
    MoveL Target_1040,v100,z5,Marcador_Data\WObj:=Tablero;
    MoveL Target_1050,v100,z5,Marcador_Data\WObj:=Tablero;
    MoveL Target_1060,v100,z5,Marcador_Data\WObj:=Tablero;
    MoveL Target_1070,v100,z5,Marcador_Data\WObj:=Tablero;
    MoveL Target_1080,v100,z5,Marcador_Data\WObj:=Tablero;
    MoveL Target_1090,v100,z5,Marcador_Data\WObj:=Tablero;
    MoveL Target_1100,v100,z5,Marcador_Data\WObj:=Tablero;
    MoveL Target_1110,v100,z5,Marcador_Data\WObj:=Tablero;
    MoveL Target_1120,v100,z5,Marcador_Data\WObj:=Tablero;
    MoveL Target_1130,v100,z5,Marcador_Data\WObj:=Tablero;
  ENDPROC
  PROC Path_110()
    MoveL Target_1140,v100,z5,Marcador_Data\WObj:=Tablero;
    MoveL Target_1150,v100,z5,Marcador_Data\WObj:=Tablero;
    MoveL Target_1160,v100,z5,Marcador_Data\WObj:=Tablero;
    MoveL Target_1170,v100,z5,Marcador_Data\WObj:=Tablero;
    MoveL Target_1180,v100,z5,Marcador_Data\WObj:=Tablero;
    MoveL Target_1190,v100,z5,Marcador_Data\WObj:=Tablero;
    MoveL Target_1200,v100,z5,Marcador_Data\WObj:=Tablero;
    MoveL Target_1210,v100,z5,Marcador_Data\WObj:=Tablero;
    MoveL Target_1220,v100,z5,Marcador_Data\WObj:=Tablero;
    MoveL Target_1230,v100,z5,Marcador_Data\WObj:=Tablero;
    MoveL Target_1240,v100,z5,Marcador_Data\WObj:=Tablero;
    MoveL Target_1250,v100,z5,Marcador_Data\WObj:=Tablero;
    MoveL Target_1260,v100,z5,Marcador_Data\WObj:=Tablero;
    MoveL Target_1270,v100,z5,Marcador_Data\WObj:=Tablero;
    MoveL Target_1280,v100,z5,Marcador_Data\WObj:=Tablero;
  ENDPROC
  PROC Path_120()
    MoveL Target_1290,v100,z5,Marcador_Data\WObj:=Tablero;
    MoveL Target_1300,v100,z5,Marcador_Data\WObj:=Tablero;
    MoveL Target_1310,v100,z5,Marcador_Data\WObj:=Tablero;
    MoveL Target_1320,v100,z5,Marcador_Data\WObj:=Tablero;
    MoveL Target_1330,v100,z5,Marcador_Data\WObj:=Tablero;
    MoveL Target_1340,v100,z5,Marcador_Data\WObj:=Tablero;
    MoveL Target_1350,v100,z5,Marcador_Data\WObj:=Tablero;
    MoveL Target_1360,v100,z5,Marcador_Data\WObj:=Tablero;
    MoveL Target_1370,v100,z5,Marcador_Data\WObj:=Tablero;
  ENDPROC
  PROC Path_130()
    MoveL Target_10,v100,z5,Marcador_Data\WObj:=Tablero;
  ENDPROC
  PROC Path_10()
    MoveAbsJ JointTarget_1,v300,z10,Marcador_Data\WObj:=Tablero;
  ENDPROC
  PROC Path_60()
    MoveL Target_1380,v100,z5,Marcador_Data\WObj:=Tablero;
    MoveL Target_1390,v100,z5,Marcador_Data\WObj:=Tablero;
    MoveL Target_1400,v100,z5,Marcador_Data\WObj:=Tablero;
    MoveL Target_1410,v100,z5,Marcador_Data\WObj:=Tablero;
  ENDPROC
  PROC Path_80()
    MoveL Target_1420,v100,z5,Marcador_Data\WObj:=Tablero;
    MoveL Target_1430,v100,z5,Marcador_Data\WObj:=Tablero;
    MoveL Target_1440,v100,z5,Marcador_Data\WObj:=Tablero;
    MoveL Target_1450,v100,z5,Marcador_Data\WObj:=Tablero;
  ENDPROC
  PROC Path_140()
    MoveAbsJ JointTarget_2,v300,z5,Marcador_Data\WObj:=Tablero;
  ENDPROC
ENDMODULE

